{attribute 'GeneratedUsingTerminal: EL3483-0060-0018'}
{attribute addProperty BoxType "EL3483-0060-0018"}
{attribute addProperty Id "VoltageAT %I*REAL4"}
{attribute addProperty CRC "2671734600"}
{attribute addProperty Size "4"}
TYPE L3_Basic_9F3F6F48 :
STRUCT
	{attribute addProperty Name "Voltage"}
	Voltage AT %I* : REAL;
END_STRUCT
END_TYPE

(* stored: Version 1.2.0.0, ProductVersion 3.1.4024.9
   DUT L3_Basic_9F3F6F48: Id {6026c995-8c5f-4cf7-a65f-78b6c021b83e} *)
